Staubli VAL3: clkValve7.pgx

program clkValve7()
begin
  call toggleValve(7)
end
